// TIA Portal V19 export
TYPE "MatCountCIn"
// stored: Access Published
   STRUCT
      Rst : Bool;
      Standstill : Bool;
      CheckNextFeeding : Bool;
      EncoderValid : Bool;
      EncoderPosValid : Bool;
      PresetExe : Bool;
      PresetPosition : LReal;
      AxisPos : LReal;
      AxisModule : LReal;
   END_STRUCT;
END_TYPE
